FUNCTION_BLOCK ByteBuffer implements I_Buffer
VAR_INPUT
END_VAR
VAR_OUTPUT
END_VAR
VAR
	buffer : POINTER TO BYTE;
	bufferSize : UDINT;
	_size : UDINT;
END_VAR
VAR CONSTANT
	SIZE_OF_INT		: UDINT := SIZEOF(INT);
	SIZE_OF_ULINT	: UDINT := SIZEOF(ULINT);
	SIZE_OF_CHAR	: UDINT := SIZEOF(BYTE);
	SIZE_OF_BOOL	: UDINT := SIZEOF(BOOL);	
END_VAR

METHOD PUBLIC AddBoolToBuffer : BOOL
VAR_IN_OUT
	Field : BOOL;
END_VAR
IF Remaining >= SIZE_OF_BOOL THEN
	
	memcpy(GetNextAvailableAddress(),ADR(Field),SIZE_OF_BOOL);
	UpdateUsedBufferSize(SIZE_OF_BOOL);

END_IF
END_METHOD

METHOD PUBLIC AddCharToBuffer : BOOL
VAR_IN_OUT
	Field : BYTE;
END_VAR
IF Remaining >= SIZE_OF_CHAR THEN
	
	memcpy(GetNextAvailableAddress(),ADR(Field),SIZE_OF_CHAR);
	UpdateUsedBufferSize(SIZE_OF_CHAR);

END_IF
END_METHOD

METHOD PUBLIC AddIntToBuffer : BOOL
VAR_IN_OUT
	Field : INT;
END_VAR
IF Remaining >= SIZE_OF_INT THEN
	
	memcpy(GetNextAvailableAddress(),ADR(Field),SIZE_OF_INT);
	UpdateUsedBufferSize(SIZE_OF_INT);

END_IF
END_METHOD

PROPERTY PUBLIC Address : pointer to byte
GET
Address := buffer;
END_GET
END_PROPERTY

METHOD PUBLIC AddStringToBuffer : BOOL
VAR_IN_OUT
	stringToWrite : STRING;
END_VAR
VAR
	sizeInBytes : UDINT;
END_VAR
sizeInBytes := INT_TO_UDINT(len(stringToWrite));

IF Remaining >= sizeInBytes THEN
	
	memcpy(GetNextAvailableAddress(),ADR(stringToWrite),sizeInBytes);
	UpdateUsedBufferSize(sizeInBytes);

END_IF
END_METHOD

METHOD PUBLIC AddULintToBuffer : BOOL
VAR_IN_OUT
	Field : ULINT;
END_VAR
IF Remaining >= SIZE_OF_ULINT THEN
	
	memcpy(GetNextAvailableAddress(),ADR(Field),SIZE_OF_ULINT);
	UpdateUsedBufferSize(SIZE_OF_ULINT);

END_IF
END_METHOD

METHOD FB_init : BOOL
VAR_INPUT
	bInitRetains : BOOL; // if TRUE, the retain variables are initialized (warm start / cold start)
	bInCopyCode : BOOL;  // if TRUE, the instance afterwards gets moved into the copy code (online change)
	Buffer : POINTER TO BYTE;
	BufferSize : UDINT;
END_VAR
THIS^.buffer := Buffer;
THIS^.bufferSize := BufferSize;
END_METHOD

METHOD PRIVATE GetNextAvailableAddress : POINTER TO BYTE
VAR_INPUT
END_VAR
GetNextAvailableAddress := buffer + _size;
END_METHOD

PROPERTY PUBLIC Remaining : UDINT
GET
Remaining := bufferSize - _size;
END_GET
END_PROPERTY

METHOD PUBLIC Reset
VAR_INPUT
END_VAR
memset(buffer,16#00,bufferSize);
_size := 0;
END_METHOD

PROPERTY PUBLIC Size : udint
GET
Size := _size;
END_GET
END_PROPERTY

METHOD PRIVATE UpdateUsedBufferSize : BOOL;
VAR_INPUT
	insertFieldSize : UDINT;
END_VAR
_size := _size + insertFieldSize;
END_METHOD

END_FUNCTION_BLOCK

(* stored: Version 1.1.0.1, ProductVersion 3.1.4024.4
   POU ByteBuffer: Id {ca8ea944-d046-45e5-b155-b381399eb26d}, SpecialFunc None
   Folder Constructor: Id {f0968fc2-fc0d-44fe-be8b-44b75a39c838}
   Folder Private: Id {cfd5ed12-5823-4495-915f-12c58331bc17}
   Method AddBoolToBuffer: Id {8dccb7f1-8d67-489f-92f7-a6df0d14b2bb}
   Method AddCharToBuffer: Id {671128d9-0a34-4dbc-a1ee-cc6932787bd4}
   Method AddIntToBuffer: Id {315b64f8-72ec-4188-b220-e8c371d2e51f}
   Property Address: Id {08b65846-8cf4-4a7b-b000-b754fee610e5}
   Get Get: Id {919393ce-229f-4d84-97b7-17b4f026bd88}
   Method AddStringToBuffer: Id {37fb52de-0739-4426-962e-e6e17dd1c605}
   Method AddULintToBuffer: Id {bf889ffa-2947-421c-8776-91fc782d14d4}
   Method FB_init: Id {cf43c425-3be4-446f-9f8f-57089e465a3e}
   Method GetNextAvailableAddress: Id {7769c87c-9b54-413e-a025-6ad3aa9cda6a}
   Property Remaining: Id {1a1cc13e-747d-42e2-bbcf-b121786faace}
   Get Get: Id {8c896a63-381c-4b8f-8619-2357686d18ab}
   Method Reset: Id {d01948c5-7dcb-4805-8b51-b51999861ba6}
   Property Size: Id {c5137921-4056-43a5-a079-2e7f36bdcc8b}
   Get Get: Id {a40168a9-d629-4640-a880-8cece7683cce}
   Method UpdateUsedBufferSize: Id {017832bc-629a-4cd8-99e8-0fe0fd8dbb32} *)
